KUKA KRL program: vw_bu_user_conf.src, vw_bu_user_conf.dat

--- vw_bu_user_conf.src ---
&ACCESS RVO
&REL 51
&COMMENT KS 2.6
&PARAM DISKPATH = VW_User/Applikation/VW_BU
&PARAM TPVW_VERSION = 8.1.8
&PARAM EDITMASK = vw_bu_user_conf
DEF vw_bu_user_conf( )
;
;*---------------------------------------------*
;* VW_Buersten                                 *
;* Version 1.0     / VKRC 4                    *
;* Bearbeitet am:                              *
;* 05.06.2015 BM neu erstellt                  *
;*---------------------------------------------*
;
END

--- vw_bu_user_conf.dat ---
&ACCESS  RV
&COMMENT KS 2.6
&PARAM DISKPATH = VW_User/Applikation/VW_Buersten
&PARAM TPVW_VERSION = 8.1.8
&PARAM EDITMASK = vw_bu_user_conf
&REL 51
DEFDAT  vw_bu_user_conf PUBLIC
;
;FOLD BOOLS
GLOBAL BOOL F_WARN_AUS[2]
F_WARN_AUS[1]=FALSE
F_WARN_AUS[2]=FALSE
;ENDFOLD Boolean
;
;FOLD Vorwahlen
GLOBAL INT WarnWert[2]
WarnWert[1]=90
WarnWert[2]=90
GLOBAL INT Verschleiss[2]
Verschleiss[1]=98
Verschleiss[2]=98
GLOBAL INT MaxAppBu=2
;ENDFOLD Vorwahlen
;
;FOLD Eingaenge
GLOBAL INT I_BU_Rueck[2]
I_BU_Rueck[1]=2273
I_BU_Rueck[2]=2305
GLOBAL INT I_LichtSchr[2]
I_LichtSchr[1]=2275
I_LichtSchr[2]=2307
GLOBAL INT I_BU_ArbPos[2]
I_BU_ArbPos[1]=2274
I_BU_ArbPos[2]=2306
GLOBAL INT I_BU_Stoer[2]
I_BU_Stoer[1]=2279
I_BU_Stoer[2]=2311
;
GLOBAL INT I_OHNE_BU[2]
I_OHNE_BU[1]=193
I_OHNE_BU[2]=201
GLOBAL INT I_MESSEN_BU[2]
I_MESSEN_BU[1]=194
I_MESSEN_BU[2]=202
GLOBAL INT I_ANW_BU[2]
I_ANW_BU[1]=195
I_ANW_BU[2]=203
GLOBAL INT I_GEWECH_BU[2]
I_GEWECH_BU[1]=196
I_GEWECH_BU[2]=204
GLOBAL INT I_REF_F_BU[2]
I_REF_F_BU[1]=197
I_REF_F_BU[2]=205
GLOBAL INT I_RES_BU[2]
I_RES_BU[1]=198
I_RES_BU[2]=206
;ENDFOLD Eingaenge
;
;FOLD Ausgaenge
GLOBAL INT O_ProzAktBu[2]
O_ProzAktBu[1]=193
O_ProzAktBu[2]=201
GLOBAL INT O_MessAktBu[2]
O_MessAktBu[1]=194
O_MessAktBu[2]=202
GLOBAL INT O_90_WARN[2]
O_90_WARN[1]=195
O_90_WARN[2]=203
GLOBAL INT O_98_STANDZ[2]
O_98_STANDZ[1]=196
O_98_STANDZ[2]=204
GLOBAL INT O_STOER_MES[2]
O_STOER_MES[1]=198
O_STOER_MES[2]=206
GLOBAL INT O_STOER_FU[2]
O_STOER_FU[1]=199
O_STOER_FU[2]=207
GLOBAL INT O_BU_STOER[2]
O_BU_STOER[1]=200
O_BU_STOER[2]=208
GLOBAL INT O_REGLSP_BU[2]
O_REGLSP_BU[1]=2276
O_REGLSP_BU[2]=2308
GLOBAL INT O_SCHNSTP_BU[2]
O_SCHNSTP_BU[1]=2277
O_SCHNSTP_BU[2]=2309
GLOBAL INT O_BU_EIN[2]
O_BU_EIN[1]=2278
O_BU_EIN[2]=2310
GLOBAL INT O_BU_RES[2]
O_BU_RES[1]=2279
O_BU_RES[2]=2311
;ENDFOLD Ausgaenge
;
;FOLD Flags
GLOBAL INT F_VW_BU[2]
F_VW_BU[1]=651
F_VW_BU[2]=661
GLOBAL INT F_MOT_ON[2]
F_MOT_ON[1]=652
F_MOT_ON[2]=662
GLOBAL INT F_VER_AUS[2]
F_VER_AUS[1]=654
F_VER_AUS[2]=664
GLOBAL INT F_FEHLM_AUS[2]
F_FEHLM_AUS[1]=655
F_FEHLM_AUS[2]=665
GLOBAL INT F_BU_STOER[2]
F_BU_STOER[1]=656
F_BU_STOER[2]=666
GLOBAL INT F_Uebw_Arbpos[2]
F_Uebw_Arbpos[1]=657
F_Uebw_Arbpos[2]=667
GLOBAL INT F_ZykMessBu[2]
F_ZykMessBu[1]=658
F_ZykMessBu[2]=668
GLOBAL INT F_m_ACF=659 ;mit ACF
;ENDFOLD Flags
;
;FOLD ZAEHLER
GLOBAL INT Z_n_bu[2]
Z_n_bu[1]=50
Z_n_bu[2]=55
GLOBAL INT Z_p_bu[2]
Z_p_bu[1]=51
Z_p_bu[2]=56
GLOBAL INT Z_UabsMinBu[2]
Z_UabsMinBu[1]=52
Z_UabsMinBu[2]=57
GLOBAL INT Z_Zmess_bu[2]
Z_Zmess_bu[1]=53
Z_Zmess_bu[2]=58
GLOBAL INT Z_StdMax_Bu[2]
Z_StdMax_Bu[1]=54
Z_StdMax_Bu[2]=59
;ENDFOLD ZAEHLER
;
;FOLD ANALOGEIN/-AUSGABEN
GLOBAL INT AO_p_bu[2]
AO_p_bu[1]=13
AO_p_bu[2]=15
GLOBAL INT AO_n_bu[2]
AO_n_bu[1]=14
AO_n_bu[2]=16
;ENDFOLD ANALOGEIN/-AUSGABEN
;
;FOLD REALS
GLOBAL REAL g_ana_n
GLOBAL REAL g_ana_p
GLOBAL REAL con_p_out
GLOBAL REAL con_n_out
GLOBAL REAL con_cnt_p
GLOBAL REAL con_cnt_n
GLOBAL REAL MAX_WEG=200.0
GLOBAL REAL Max_Verschleiss=100.0
;
GLOBAL REAL dm_min[2]
dm_min[1]=200.0
dm_min[2]=200.0
;
GLOBAL REAL dm_max[2]
dm_max[1]=200.0
dm_max[2]=200.0
;
GLOBAL REAL dm_akt[2]
dm_akt[1]=199.0
dm_akt[2]=199.0
;
GLOBAL REAL suchweg[2]
suchweg[1]=50.0
suchweg[2]=50.0
;
GLOBAL INT v_nenn[2]
v_nenn[1]=1490
v_nenn[2]=1490
;
GLOBAL INT v_d_min[2]
v_d_min[1]=3000
v_d_min[2]=3000
;
GLOBAL INT v_d_max[2]
v_d_max[1]=3000
v_d_max[2]=3000
;
GLOBAL REAL u_dmin[2]
u_dmin[1]=100.0
u_dmin[2]=100.0
;
GLOBAL REAL u_dmax[2]
u_dmax[1]=100.0
u_dmax[2]=100.0
;ENDFOLD REALS
;
;FOLD FRAMES
GLOBAL FRAME REF_POS[2]
REF_POS[1]={X -108.30928,Y -3105.38745,Z 508.149994,A -53.717701,B 89.99823,C 126.28083}
REF_POS[2]={X -108.305565,Y -3105.37866,Z 505.285675,A -66.6040955,B 89.9970779,C 113.39402}
;
GLOBAL FRAME MESS_POS[2]
MESS_POS[1]={X -108.313927,Y -3105.3606,Z 464.777893,A 108.71019,B 89.9989624,C -71.2901077}
MESS_POS[2]={X -108.313835,Y -3105.3606,Z 464.77771,A 108.725204,B 89.9989395,C -71.2751007}
;ENDFOLD FRAMES
ENDDAT
